PROGRAM main
  VAR
    At_Entry AT %IX0.0 : BOOL;
    Low_Box AT %IX0.1 : BOOL;
    High_Box AT %IX0.2 : BOOL;
    At_Turntable_Entry AT %IX0.3 : BOOL;
    At_Load_Position AT %IX0.4 : BOOL;
    At_Unload_Position AT %IX0.5 : BOOL;
    At_Front AT %IX0.6 : BOOL;
    At_Right_Entry AT %IX0.7 : BOOL;
    At_Left_Entry AT %IX1.0 : BOOL;
    At_Right_Exit AT %IX1.1 : BOOL;
    At_Left_Exit AT %IX1.2 : BOOL;
    Start_Button AT %IX1.3 : BOOL;
    Reset_Button AT %IX1.4 : BOOL;
    Stop_Button AT %IX1.5 : BOOL;
    Emergency_Stop AT %IX1.6 : BOOL;
    Auto_Mode AT %IX1.7 : BOOL;
    Feeder_Conveyor AT %QX0.0 : BOOL;
    Entry_Conveyor AT %QX0.1 : BOOL;
    Load AT %QX0.2 : BOOL;
    Unload AT %QX0.3 : BOOL;
    Turn AT %QX0.4 : BOOL;
    Left_Conveyor AT %QX0.5 : BOOL;
    Right_Conveyor AT %QX0.6 : BOOL;
    Green_Indicator AT %QX0.7 : BOOL;
    Yellow_Indicator AT %QX1.0 : BOOL;
    Red_Indicator AT %QX1.1 : BOOL;
    Start_Light AT %QX1.2 : BOOL;
    Reset_Light AT %QX1.3 : BOOL;
    Stop_Light AT %QX1.4 : BOOL;
    Counter AT %QW0 : INT;
    Fault_Latch : BOOL;
    System_Run : BOOL;
    S0_Idle : BOOL;
    S1_Transport : BOOL;
    S2_Load : BOOL;
    S3_Turn : BOOL;
    S4_Unload : BOOL;
    S5_Delivered : BOOL;
    Box_Tall : BOOL;
    Box_Short : BOOL;
    Height_OK : BOOL;
    Side_Entry_Det : BOOL;
    Side_Seen : BOOL;
    T_Turn : TON;
    T_Return : TON;
    T_Load_Delay : TON;
    T_Side_Delay : TON;
    C_Boxes : CTU;
  END_VAR

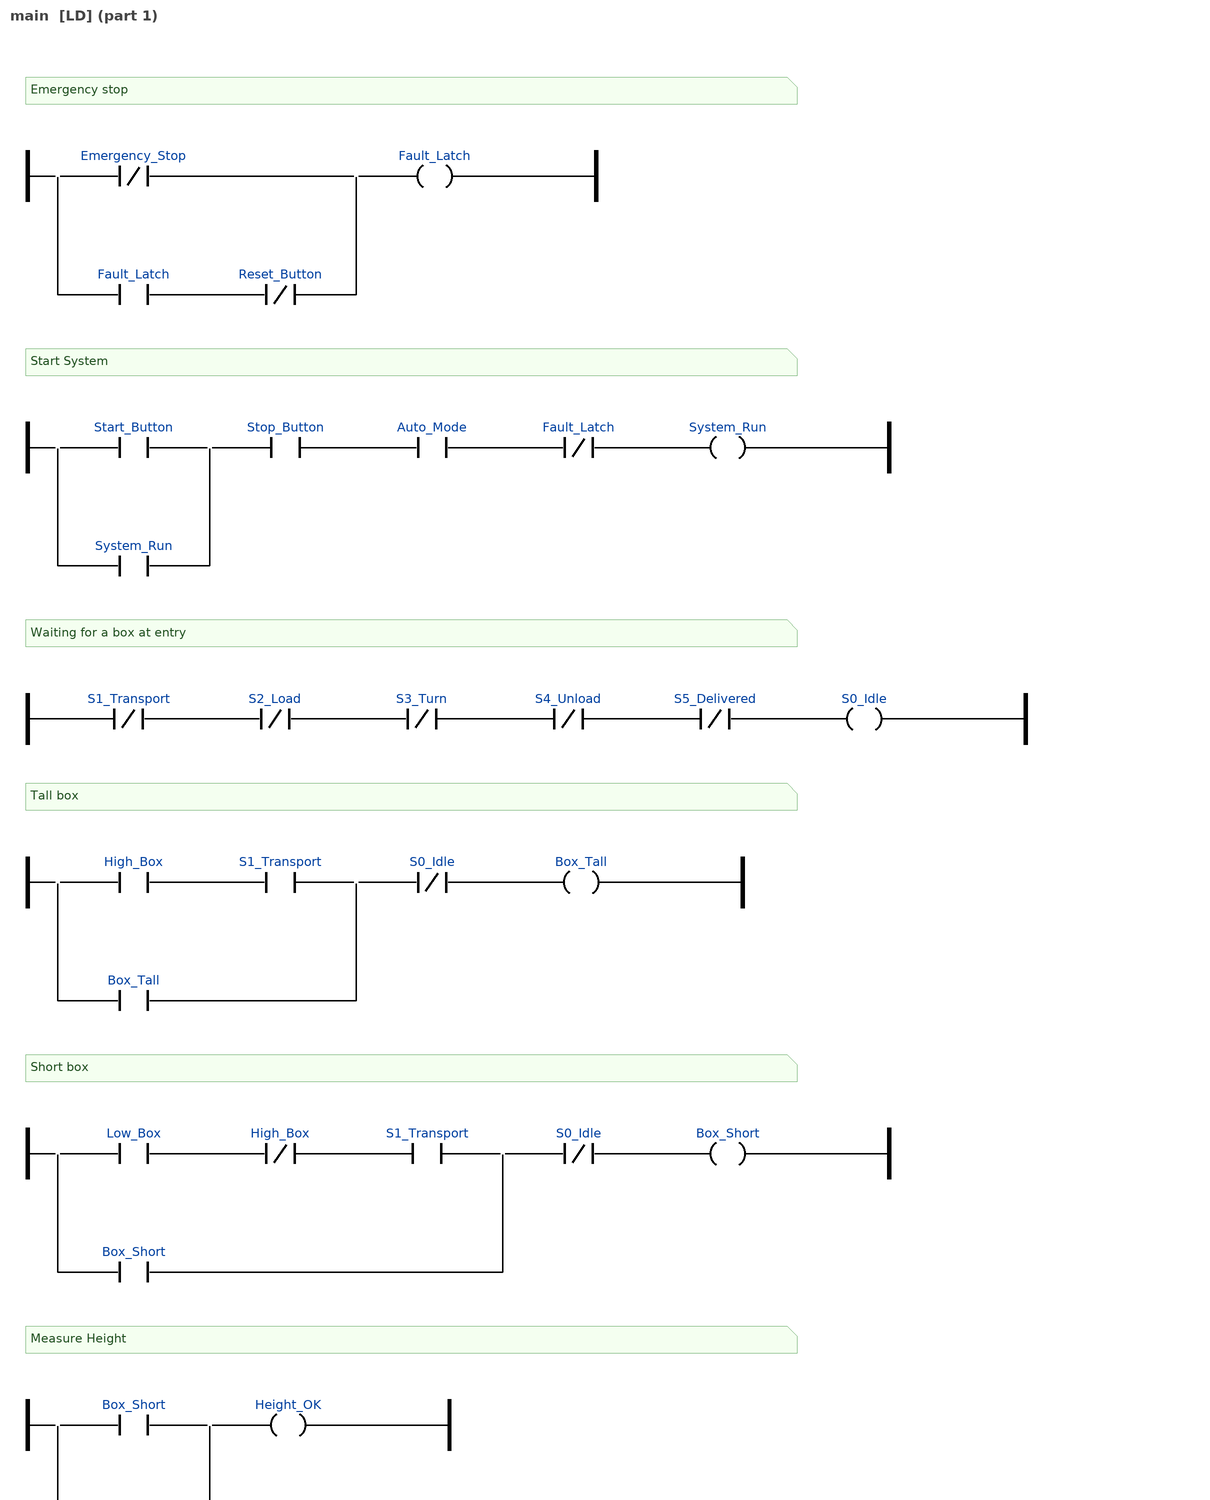
(* LD diagram, written out as Structured Text *)
(* Emergency stop *)
Fault_Latch := NOT Emergency_Stop OR Fault_Latch AND NOT Reset_Button;
(* Start System *)
System_Run := (Start_Button OR System_Run) AND Stop_Button AND Auto_Mode AND NOT Fault_Latch;
(* Waiting for a box at entry *)
S0_Idle := NOT S1_Transport AND NOT S2_Load AND NOT S3_Turn AND NOT S4_Unload AND NOT S5_Delivered;
(* Tall box *)
Box_Tall := (High_Box AND S1_Transport OR Box_Tall) AND NOT S0_Idle;
(* Short box *)
Box_Short := (Low_Box AND NOT High_Box AND S1_Transport OR Box_Short) AND NOT S0_Idle;
(* Measure Height *)
Height_OK := Box_Short OR Box_Tall;
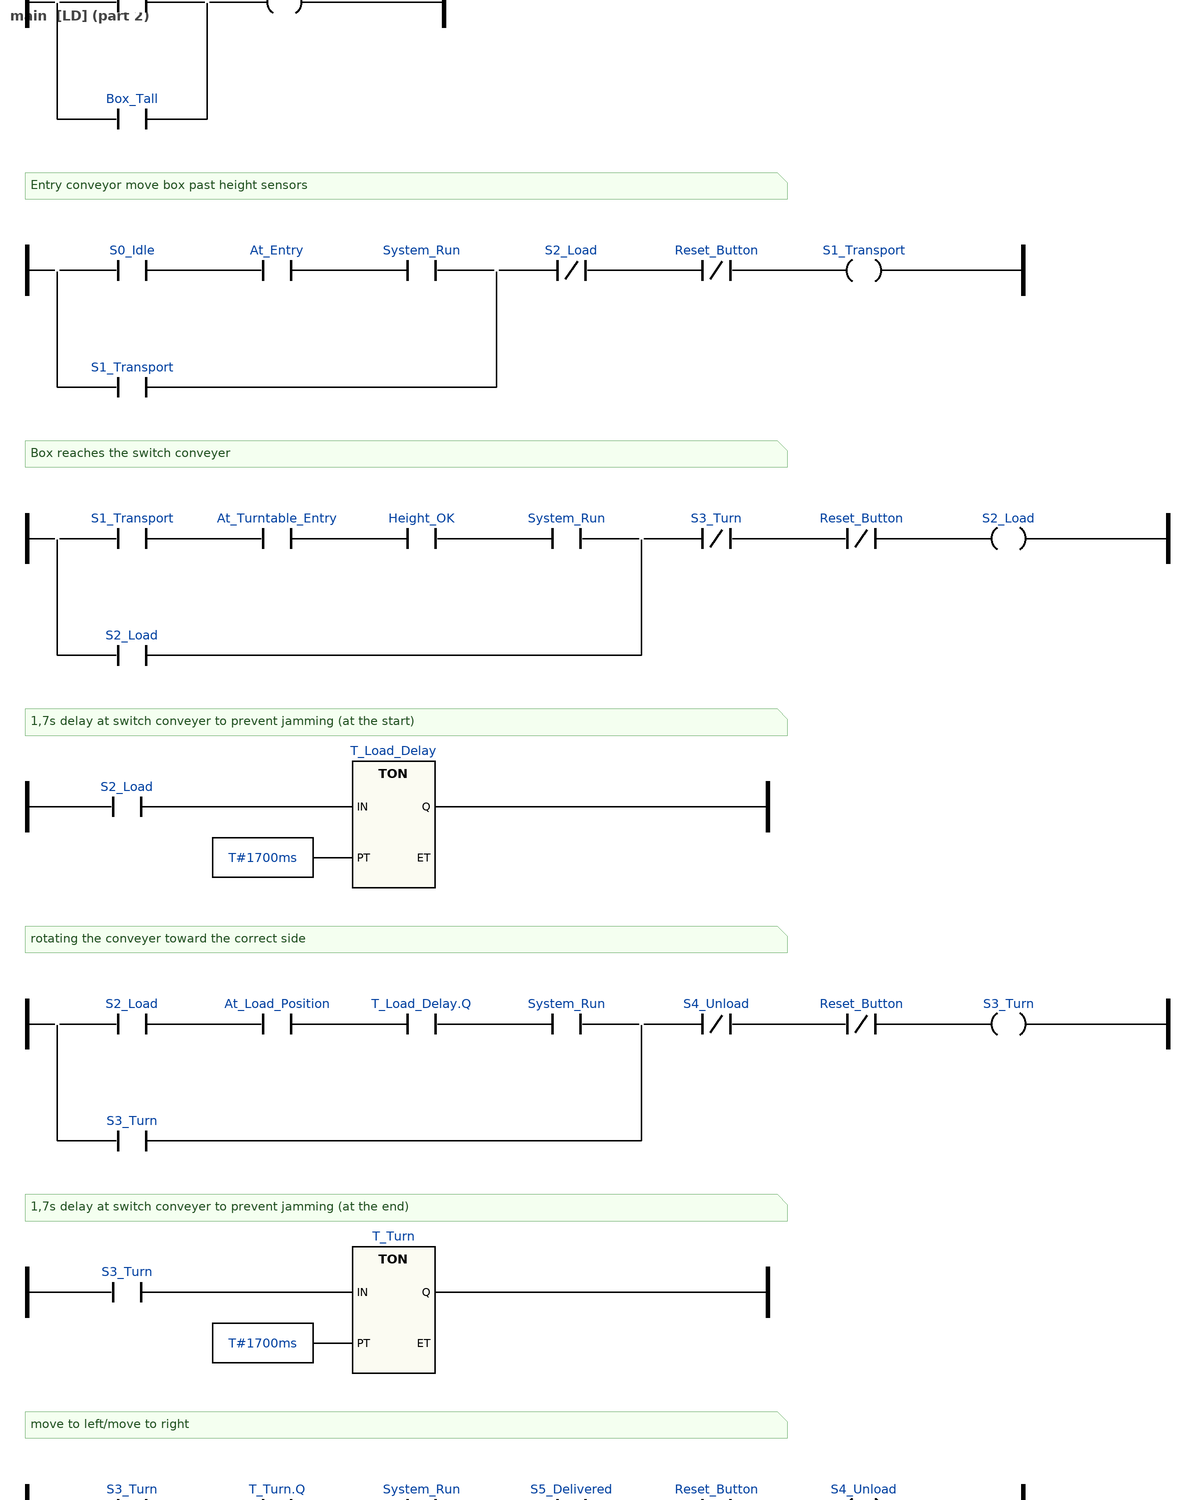
(* Entry conveyor move box past height sensors *)
S1_Transport := (S0_Idle AND At_Entry AND System_Run OR S1_Transport) AND NOT S2_Load AND NOT Reset_Button;
(* Box reaches the switch conveyer *)
S2_Load := (S1_Transport AND At_Turntable_Entry AND Height_OK AND System_Run OR S2_Load) AND NOT S3_Turn AND NOT Reset_Button;
(* 1,7s delay at switch conveyer to prevent jamming (at the start) *)
(* rotating the conveyer toward the correct side *)
S3_Turn := (S2_Load AND At_Load_Position AND T_Load_Delay.Q AND System_Run OR S3_Turn) AND NOT S4_Unload AND NOT Reset_Button;
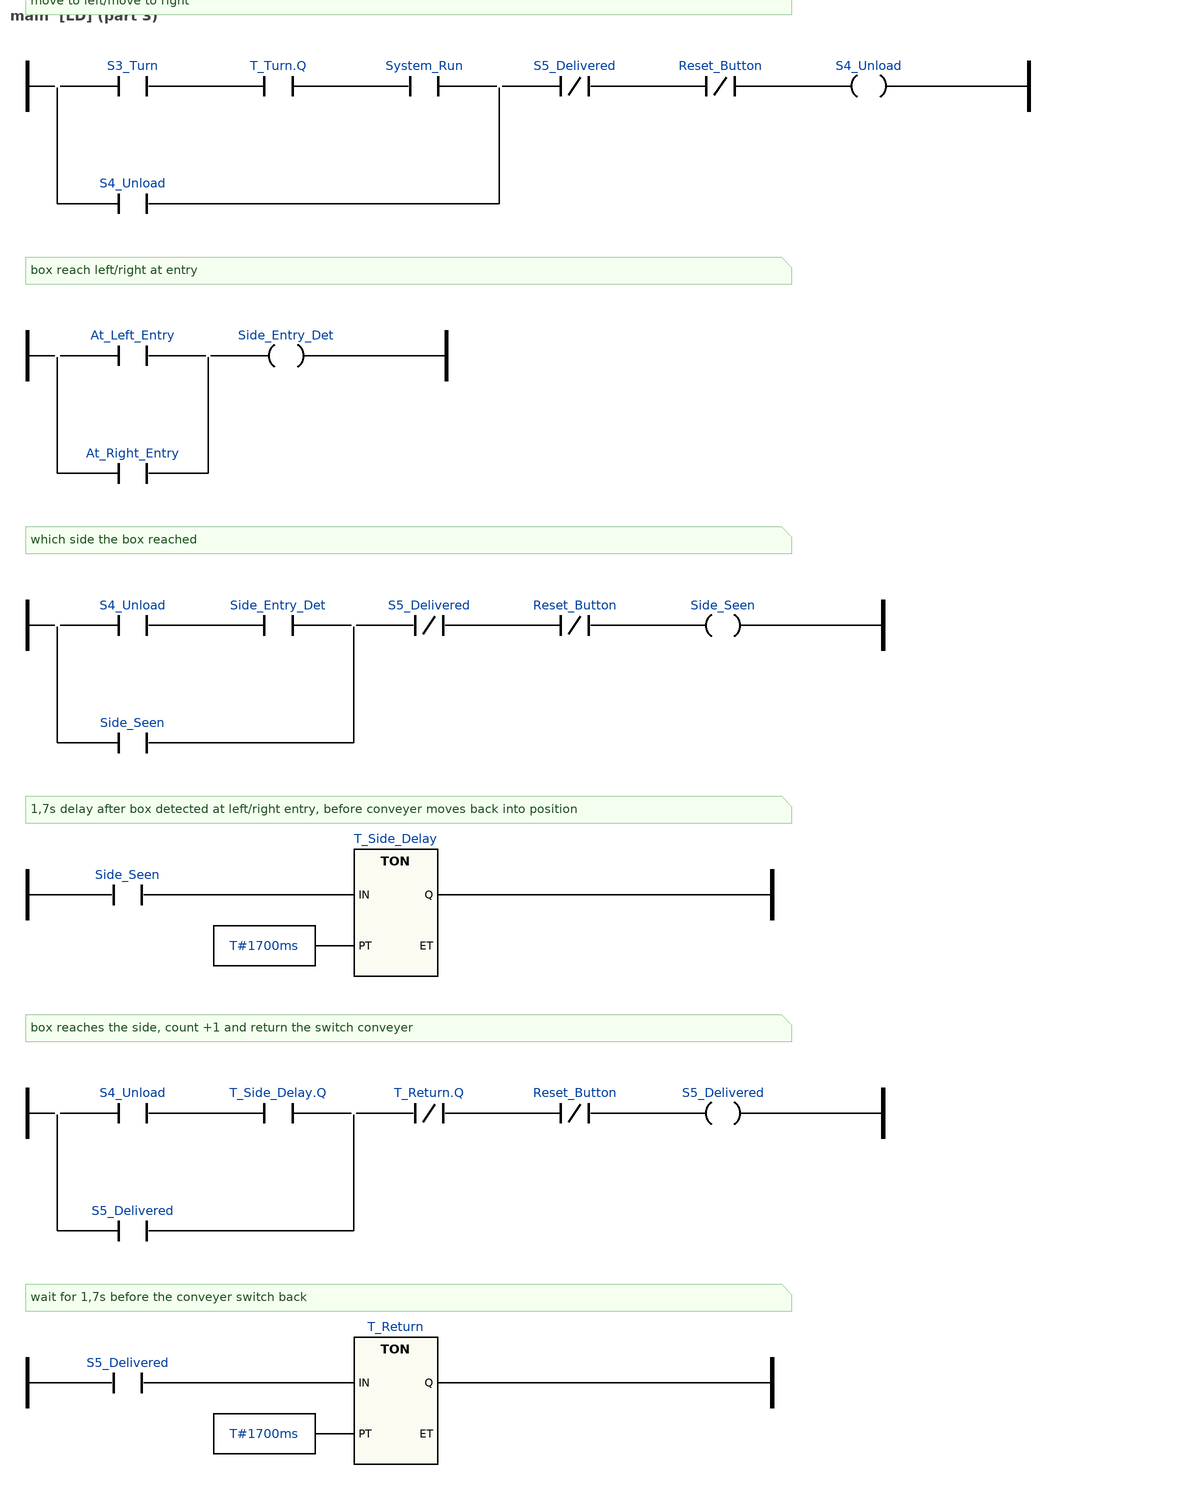
(* 1,7s delay at switch conveyer to prevent jamming (at the end) *)
(* move to left/move to right *)
S4_Unload := (S3_Turn AND T_Turn.Q AND System_Run OR S4_Unload) AND NOT S5_Delivered AND NOT Reset_Button;
(* box reach left/right at entry *)
Side_Entry_Det := At_Left_Entry OR At_Right_Entry;
(* which side the box reached *)
Side_Seen := (S4_Unload AND Side_Entry_Det OR Side_Seen) AND NOT S5_Delivered AND NOT Reset_Button;
(* 1,7s delay after box detected at left/right entry, before conveyer moves back into position *)
(* box reaches the side, count +1 and return the switch conveyer *)
S5_Delivered := (S4_Unload AND T_Side_Delay.Q OR S5_Delivered) AND NOT T_Return.Q AND NOT Reset_Button;
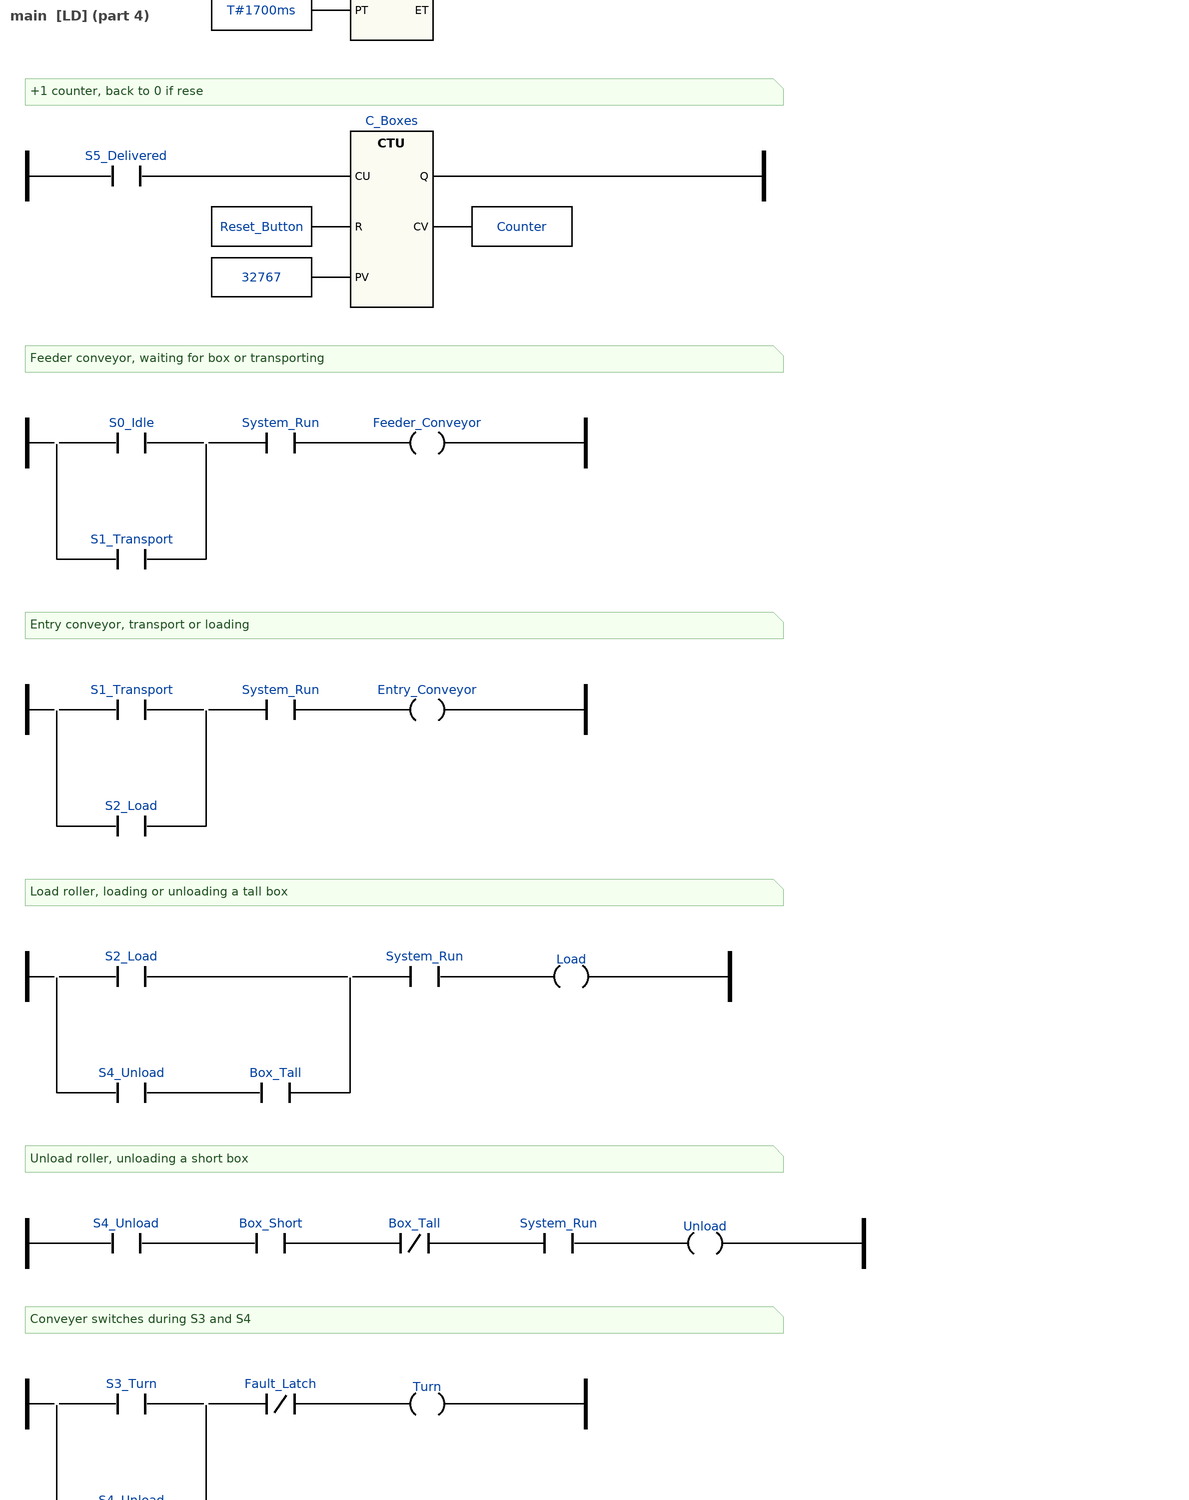
(* wait for 1,7s before the conveyer switch back *)
(* +1 counter, back to 0 if rese *)
C_Boxes(CU := S5_Delivered, R := Reset_Button, PV := 32767);
Counter := C_Boxes.CV;
(* Feeder conveyor, waiting for box or transporting *)
Feeder_Conveyor := (S0_Idle OR S1_Transport) AND System_Run;
(* Entry conveyor, transport or loading *)
Entry_Conveyor := (S1_Transport OR S2_Load) AND System_Run;
(* Load roller, loading or unloading a tall box *)
Load := (S2_Load OR S4_Unload AND Box_Tall) AND System_Run;
(* Unload roller, unloading a short box *)
Unload := S4_Unload AND Box_Short AND NOT Box_Tall AND System_Run;
(* Conveyer switches during S3 and S4 *)
Turn := (S3_Turn OR S4_Unload) AND NOT Fault_Latch;
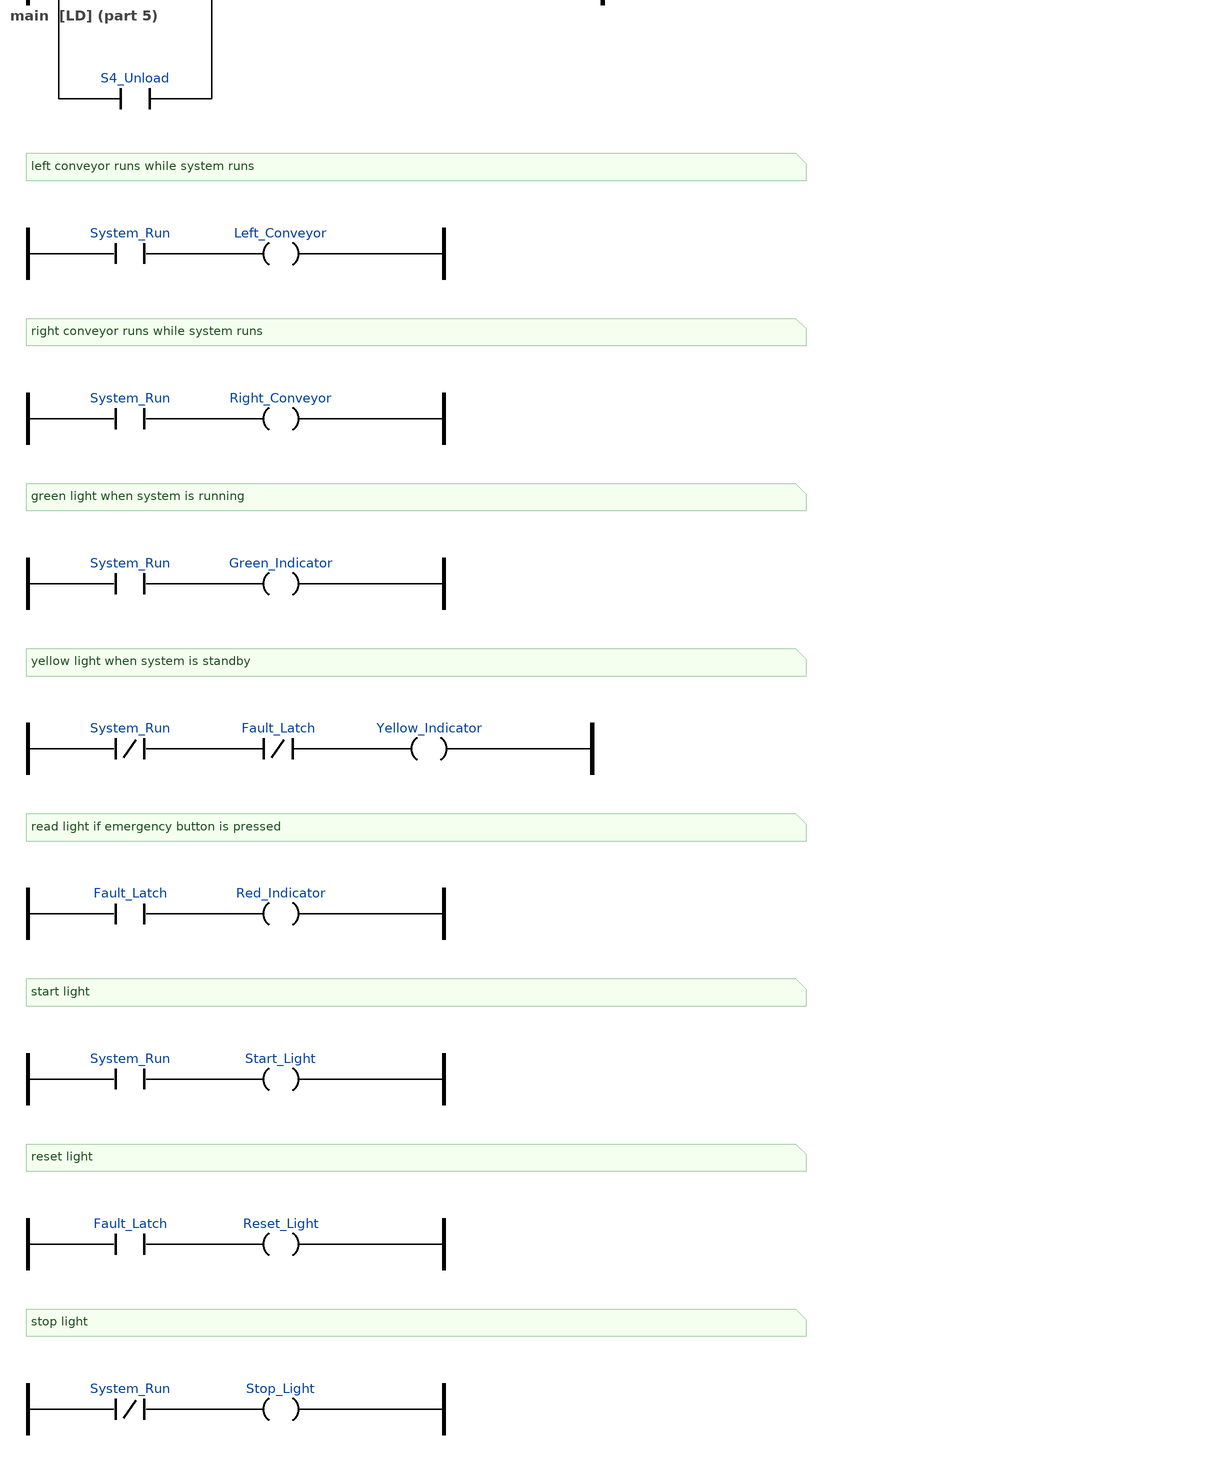
(* left conveyor runs while system runs *)
Left_Conveyor := System_Run;
(* right conveyor runs while system runs *)
Right_Conveyor := System_Run;
(* green light when system is running *)
Green_Indicator := System_Run;
(* yellow light when system is standby *)
Yellow_Indicator := NOT System_Run AND NOT Fault_Latch;
(* read light if emergency button is pressed *)
Red_Indicator := Fault_Latch;
(* start light *)
Start_Light := System_Run;
(* reset light *)
Reset_Light := Fault_Latch;
(* stop light *)
Stop_Light := NOT System_Run;
T_Load_Delay(IN := S2_Load, PT := T#1700ms);
T_Turn(IN := S3_Turn, PT := T#1700ms);
T_Side_Delay(IN := Side_Seen, PT := T#1700ms);
T_Return(IN := S5_Delivered, PT := T#1700ms);
END_PROGRAM
